(* CODESYS project EAS SCADA BATCH.library
   Company: ESCARRE AUTOMATIZACION Y SERVICIOS sl
   Description: Ajuste comunicacion ADS
      Ajuste tamaño constantes
   Version: 1.1.1
   Placeholder: EAS SCADA BATCH
   Author: EAS
   Title: EAS SCADA BATCH

Project tree, tasks and I/O mapping:
  libraries: Tc2_Standard, * (Beckhoff Automation GmbH); Tc2_System, * (Beckhoff Automation GmbH); Tc3_Module, * (Beckhoff Automation GmbH)
  DUTs/
    PE/
      data type E_Funcio
      data type PasCicle
      data type T_Compat
      data type T_funcio
      data type T_Sirena
  GVLs/
    global variables Batch
    global variables CONSTANTS
  POUs/
    BATCH/
      function block CarregarFuncionsActivesAlDB [ST]
      function block ComprobarFuncionsPas [ST]
      function block Inic_Func_Actv [ST]
      function block Parar_Func_FiFuncio [ST]
      function block Parar_Func_Incomp [ST]
      function block PararTotesLesFuncions [ST]
      function block Salt [ST]
      function block SaltDePasEnUnCicle [ST]
    GestioPE/
      function block FunBck_v01 [ST]
      function block Func_Activa_v01 [ST]
  VISUs/
*)

// DUTs/PE/E_Funcio
TYPE E_Funcio :
STRUCT

	Cd_Funcio:WORD;
	Actv_Funcio:BOOL;
	ParamFunc:ARRAY [1..Max_ParamFunc] OF WORD;

END_STRUCT
END_TYPE

// DUTs/PE/PasCicle
TYPE PasCicle :
STRUCT
	Pas:WORD;
	Funcio:E_Funcio;

END_STRUCT
END_TYPE

// DUTs/PE/T_Compat
TYPE T_Compat :
STRUCT

	Funcio1:WORD;  			(*Codi de la primera funcio*)
	Funcio2:WORD;  			(*Codi de la segona funcio*)

END_STRUCT
END_TYPE

// DUTs/PE/T_funcio
TYPE T_funcio :
STRUCT

	Cd_funcio:WORD;												(*Codi de la funció*)
	DesFuncio:STRING(16);										(*Descripció de la funció*)
	Background:BOOL;												(*Indicació per si la funció es en backgraund o no*)
	FinFunc:ARRAY [1..max_FinFunc] OF WORD;					(*Funcions que s'han d'acabar al començar aquesta*)

END_STRUCT
END_TYPE

// DUTs/PE/T_Sirena
TYPE T_Sirena :
STRUCT
	Actv:BOOL;
	Rearme:BOOL;
END_STRUCT
END_TYPE

// GVLs/Batch

VAR_GLOBAL RETAIN

(*=======================================	*)
(*					Estat del PE4							*)
(*=======================================	*)

(*Estat de PE4*)
	Func_Comp: ARRAY [1..Max_Compatibles] OF T_Compat;


(*=======================================	*)
(*			Variables de gestió de funcions				*)
(*=======================================	*)

(*Estat de lesFuncions *)
	Est_Func: ARRAY [1..Max_Funcions] OF E_Funcio;  		(*Estat actual de les funcions*)
	Est_F_PE4: ARRAY [1..Max_Funcions] OF E_Funcio;  		(*Estat de les funcions per les comunicacions del PE4*)
	Est_F_PE4_Ant: ARRAY [1..Max_Funcions] OF E_Funcio;  	(*Estat de les funcions per les comunicacions del PE4*)


(* *)
	Config_Func: ARRAY  [1..Max_Funcions] OF t_funcio;		(*Configuració de les funcios *)
	Func_Actives: ARRAY [1..Max_Func_Pas] OF WORD;		(* DB que indica en automaatic les funcions que estan en marcha en automatic*)


(*=======================================	*)
(*			Variables de gestió de cicle					*)
(*=======================================	*)

(*Cicles*)
	Cicle0: ARRAY [1..max_PasCicle] OF PasCicle;  			(*Cicle Actual de treball*)
	CicleRebut: ARRAY [1..max_PasCicle] OF PasCicle;  		(*Cicle Rebut*)


	

(*=======================================	*)
(*			Botons Auto/Man								*)
(*=======================================	*)

	PulsadorManual:BOOL;
	PulsadorAutomatic:BOOL;

(*=======================================	*)
(*			Marcas Internes								*)
(*=======================================	*)

	InicioCiclo:BOOL;


END_VAR


VAR_GLOBAL

(*=======================================	*)
(*			Maquina paralel 								*)
(*=======================================	*)

	TipoParalelo:WORD;
	MaquinaEnParalel:BOOL:=FALSE;
	Master:BOOL;
	Slave:BOOL;
	Pas_M:DWORD;
	Pas_S1:DWORD;
	Pas_S2:DWORD;
	Pas_S3:DWORD;
	Pas_S4:DWORD;
	Tipus_P:DWORD;
	Preparat_C_local:BOOL;
	He_C_local:BOOL;
	Ordre_C:BOOL;
	Ordre_C_Master:BOOL;
	Preparat_C_S1:BOOL;
	Preparat_C_S2:BOOL;
	Preparat_C_S3:BOOL;
	Preparat_C_S4:BOOL;
	He_C_S1:BOOL;
	He_C_S2:BOOL;
	He_C_S3:BOOL;
	He_C_S4:BOOL;
	Fi_C:BOOL;
	Fi_C_master:BOOL;



(*			CONSERVAR  COMPATIBILITAT				*)

	EsperaParalelPerSaltar:BOOL;
	SaltdePas:BOOL;


END_VAR

// GVLs/CONSTANTS

VAR_GLOBAL CONSTANT

(*=======================================	*)
(*			Carregar Constants						*)
(*=======================================	*)
	Max_Funcions:WORD:=128;
	Max_ParamFunc:WORD:=9;
	max_FinFunc:WORD:=5;
	max_PasCicle:WORD:=256;
	Max_Compatibles:WORD:=32;
	Max_Func_Pas:WORD:=12;

END_VAR


(*********************************************************************


	Max_ParamFixes:WORD:=150;
	Max_DBFiFuncio: WORD:=640 ;				(* Es calcula com    (Max_Funcions*Max_FinFunc)   *)
	Max_ElementsCicle: WORD:=2816 ;		(* Es calcula com    (Max_PasCicle*(Max_ParamFunc+2))  *)
	Max_DBIncompatibles: WORD:=128;			(* Es calcula com    (Max_Compatibles*2)  *)
	Max_Inputs: WORD:=128;
	Max_Outputs: WORD:=128;
	Max_Analog: WORD:=128;
	Num_Prod_Dos:WORD:=10;         					(* Numero maximo de productos en una dosificación*)
	Max_Prod_Dos:WORD:=128;							(* Productos en una dosificadora*)
	Max_Valv_Dos:WORD:=128;							(* Valvulas en una dosificadora*)
	Max_Alarmes:WORD:=128;



***************************************************************************)

// POUs/BATCH/CarregarFuncionsActivesAlDB
FUNCTION_BLOCK CarregarFuncionsActivesAlDB

(***********************************************************************
Aquest Bloc Carrega les Funcions actives al "DB d'estat de les funcions"
al "DB de funcions actives".   
************************************************************************)

VAR_INPUT
	EstatFuncions: ARRAY [1..max_funcions] OF E_Funcio;
END_VAR

VAR_OUTPUT
	FuncionsActives:ARRAY [1..Max_Func_Pas] OF WORD;
END_VAR

VAR
	Punter:WORD;
	PunterDB:WORD;
	inicialitzaDB: Inic_Func_Actv;
	DB_ple: BOOL;

END_VAR

inicialitzaDB(Func_Actv:= FuncionsActives);
DB_Ple:=FALSE;
punter:=1;
punterDB:=1;
WHILE (punter<=max_funcions)AND NOT(DB_Ple)
	DO
		IF EstatFuncions[punter].Actv_Funcio
			THEN
				FuncionsActives[PunterDB]:=EstatFuncions[punter].Cd_Funcio;
				PunterDB:=PunterDB+1;
				IF punterDB>Max_Func_Pas
					THEN
						DB_ple:=TRUE;
				END_IF
		END_IF
		punter:=punter+1;
END_WHILE

END_FUNCTION_BLOCK

// POUs/BATCH/Inic_Func_Actv
FUNCTION_BLOCK Inic_Func_Actv

(*********************************************************
Reinicia el DB de les funcions actives
***********************************************************)

VAR_IN_OUT
	Func_Actv: ARRAY [1..Max_Func_Pas] OF WORD;		(* DB que indica en automaatic les funcions que estan en marcha en automatic*)
END_VAR

VAR
	Punter: WORD;
END_VAR

Punter:=1;

REPEAT
	Func_Actv[punter]:=0;
	Punter:=Punter+1;
UNTIL
	Punter>Max_Func_Pas
END_REPEAT

END_FUNCTION_BLOCK

// POUs/BATCH/ComprobarFuncionsPas
FUNCTION_BLOCK ComprobarFuncionsPas

(************************************************************
Aquest Bloc Comproba les funcions actves que hi ha en aquest
pas i quan acaben dona l'ordr de canviar de pas.
**************************************************************)

VAR_INPUT
	Estat_F: ARRAY [1..Max_Funcions] OF E_Funcio;
	Tipus_F:ARRAY [1..Max_Funcions] OF T_Funcio;
	FuncionsActives:ARRAY [1..Max_Func_Pas] OF WORD;
END_VAR

VAR_OUTPUT
	AumentaPas:BOOL;
END_VAR

VAR
	Punter: WORD;
	Aumenta: BOOL;
	TempoPAS:TON;

END_VAR

(*Inicialitzar els punters*)
Punter:=1;
Aumenta:=TRUE;

REPEAT
	IF (FuncionsActives[Punter]<>0)AND((Estat_F[FuncionsActives[Punter]].Actv_Funcio=TRUE)AND(Tipus_F[FuncionsActives[Punter]].Background=FALSE))
		THEN
			Aumenta:=FALSE;
	END_IF
	Punter:=Punter+1;
UNTIL
	(Punter>Max_Func_Pas)OR(Aumenta=FALSE)
END_REPEAT

TempoPAS
	(IN:=Aumenta ,
	PT:=t#500ms ,
	Q=>AumentaPas ,
	ET=> );

END_FUNCTION_BLOCK

// POUs/BATCH/Parar_Func_FiFuncio
FUNCTION_BLOCK Parar_Func_FiFuncio

(**************************************************
Para les funcions del "DB de l'estat de funcions" 
depenen de la funcio de la entreda per "fifuncion"
***************************************************)

VAR_INPUT
	Tipus_Funcio:T_funcio;
END_VAR
VAR_OUTPUT
END_VAR
VAR_IN_OUT
	Estat_F: ARRAY [1..Max_Funcions] OF E_Funcio;
END_VAR
VAR
	PunterFiFunc:WORD;
	FuncioIncompat: WORD;
END_VAR

(*..................	Parar les funcions per fin función..................................	*)
PunterFiFunc:=1;
WHILE (PunterFiFunc <= max_FinFunc) DO
	FuncioIncompat :=Tipus_funcio.FinFunc[PunterFiFunc];
	IF FuncioIncompat <>0
		THEN
			Estat_F [FuncioIncompat].Actv_Funcio:=FALSE;
	END_IF
	PunterFiFunc:=PunterFiFunc+1;
END_WHILE

END_FUNCTION_BLOCK

// POUs/BATCH/Parar_Func_Incomp
FUNCTION_BLOCK Parar_Func_Incomp
(************************************************************
L'hi introduim una funció i el el bloc para les funcions del 
"DB estat de les funcions" depenen del 
"DB de compatibilitat"
**************************************************************)
VAR_INPUT
	Funcio:WORD;  (*Funcio que s'ha de parar*)
END_VAR

VAR_OUTPUT
END_VAR

VAR_IN_OUT
	DB_Comp:ARRAY [1..Max_Compatibles] OF T_Compat;
	Estat_F: ARRAY [1..Max_Funcions] OF E_Funcio;
END_VAR

VAR
	PunterEstat:WORD;
	PunterComp:WORD;
END_VAR

(*Mirar si hi ha alguna funció incompatible amb la nova funció*)
PunterEstat:=1;
PunterComp:=1;
REPEAT
	IF DB_Comp[PunterComp].Funcio1=Funcio
		THEN
			PunterEstat:=DB_Comp[PunterComp].Funcio2;
			Estat_F[PunterEstat].Actv_Funcio:=FALSE;
	END_IF
	PunterComp:=PunterComp+1;
UNTIL
	(PunterComp>Max_Compatibles)
END_REPEAT

END_FUNCTION_BLOCK

// POUs/BATCH/PararTotesLesFuncions
FUNCTION_BLOCK PararTotesLesFuncions
(********************************************************
Parar totes les funcions del "DB estat"
*********************************************************)
VAR_IN_OUT
	Estat_F: ARRAY [1..Max_Funcions] OF E_Funcio;
END_VAR

VAR
	Punter: WORD;
END_VAR

(*Inicialitzar els punters*)
Punter:=1;


WHILE (Punter <= Max_Funcions) DO
	IF Estat_F[Punter].Actv_Funcio=TRUE
		THEN
			Estat_F [Punter].Actv_Funcio:=FALSE;
	END_IF
	Punter:=Punter+1;
END_WHILE

END_FUNCTION_BLOCK

// POUs/BATCH/Salt
FUNCTION_BLOCK Salt
(************************************************************
Salta del "Pas inicial" al "Pas Final"  del  "BDCicle"
**************************************************************)
VAR_INPUT
	PasInicial:DWORD;
	PasFinal:DWORD;
END_VAR

VAR_IN_OUT


END_VAR

VAR

	FIFuncio:Parar_Func_FiFuncio;
	Incompatibles:Parar_Func_Incomp;
	PunterCicle:WORD;					(* Aquest valor marca la popsició del db de cicle on estem independent del pas de cicle *)
	T_Func_Act:T_Funcio;				(* Funcio que indica el punterCicle *)

	codi: WORD;

	Est_Func_0: ARRAY [1..Max_Funcions] OF E_Funcio;  		(*Estat de les funcions a cero per reiniciar l'estat*)
END_VAR

(*,,,,,,,,,,,,,,,,,,,,Carregar la posició inicial depenen si es salta desde:
				el pas cero: carerega d'un cicle nou
				un pas en concret: salt sobre el cicle que ja està carregat ,,,,,,,,,,,,,,,,,,,,,  *)

IF PasInicial=0
	THEN
		(*Posar Punter al primer pas*)
		PunterCicle:=1;
		(*Inicialitzar el estat de les funcions*)
		Est_Func:=Est_Func_0;
	ELSE
		(*Buscar Punter Cicle del pas inicial*)
		PunterCicle:=0;
		REPEAT
			PunterCicle := PunterCicle+1;
		UNTIL
			(((Cicle0[PunterCicle].Pas=PasInicial)AND(Cicle0[PunterCicle+1].Pas<>PasInicial)) OR (PunterCicle>=max_PasCicle))
		END_REPEAT
		PunterCicle := PunterCicle+1;      (*02/06/05*)
END_IF

(*,,,,,,,,,,,,,,,,,,,,Bucle de control,,,,,,,,,,,,,,,,,,,,,,,,,,,,,,,,,,,,,,,,,,,,,,,,,,,,,,,,,,,,,	*)

REPEAT
(*.................. Carregar la funció del pas............................................. *)
		codi:=Cicle0[PunterCicle].Funcio.Cd_Funcio;
		IF codi<>0 THEN
		T_Func_Act:=Config_Func[codi];
		END_IF
(*..................	Parar les funcions incompatibles..................................	*)
		Incompatibles(
			Funcio:=T_Func_Act.Cd_funcio ,
			DB_Comp:= Func_Comp ,
			Estat_F:= Est_Func );

(*..................	Activar si es en Background ........................................	*)
		IF T_Func_Act.Background=TRUE
			THEN
				Est_Func[T_Func_Act.Cd_Funcio] := Cicle0[PunterCicle].Funcio ; 	(*Carregar parametres*)
				Est_Func[T_Func_Act.Cd_Funcio].Actv_Funcio:=TRUE;			(*Posar la funció en actiu*)
		END_IF

(*..................	Parar les funcions per fin función..................................	*)
		FiFuncio(
			Tipus_Funcio:=  T_Func_Act ,
			 Estat_F:=Est_Func	 );

(*,,,,,,,,,,,,,,,,,,	Activar funció,,,,,,,,,,,,,,,,,,,,,,,,,,,,,,,,,,,,,,,,,,,,,,,,,,,,,,,,,,,,,,,,,,,	*)
		IF Cicle0[PunterCicle].Pas = PasFinal
			THEN
				Est_Func[T_Func_Act.Cd_Funcio] := Cicle0[PunterCicle].Funcio ;	(*Carregar parametres*)
				Est_Func[T_Func_Act.Cd_Funcio].Actv_Funcio := TRUE;			(*Posar la funció en actiu*)
		END_IF

(*,,,,,,,,,,,,,,,,,,Aumentar el Punter del cicle,,,,,,,,,,,,,,,,,,,,,,,,,,,,,,,,,,,,,,,,,,	*)
		PunterCicle := PunterCicle+1;

UNTIL
	(((Cicle0[PunterCicle].Pas <> PasFinal)AND(Cicle0[PunterCicle-1].Pas = PasFinal))
	OR(PunterCicle>max_PasCicle)
	OR(Cicle0[PunterCicle-1].Funcio.Cd_Funcio=0))
END_REPEAT

END_FUNCTION_BLOCK

// POUs/BATCH/SaltDePasEnUnCicle
FUNCTION_BLOCK SaltDePasEnUnCicle
(************************************************************
Salta del "Pas inicial" al "Pas Final"  del  "BDCicle"
**************************************************************)
VAR_INPUT
	PasInicial:DWORD;
	PasFinal:DWORD;
END_VAR

VAR_IN_OUT


END_VAR

VAR

	FIFuncio:Parar_Func_FiFuncio;
	Incompatibles:Parar_Func_Incomp;
	PunterCicle:WORD;					(* Aquest valor marca la popsició del db de cicle on estem independent del pas de cicle *)
	T_Func_Act:T_Funcio;				(* Funcio que indica el punterCicle *)

	codi: WORD;

	Est_Func_0: ARRAY [1..Max_Funcions] OF E_Funcio;  		(*Estat de les funcions a cero per reiniciar l'estat*)
END_VAR

(*,,,,,,,,,,,,,,,,,,,,Carregar la posició inicial depenen si es salta desde:
				el pas cero: carerega d'un cicle nou
				un pas en concret: salt sobre el cicle que ja està carregat ,,,,,,,,,,,,,,,,,,,,,  *)

IF PasInicial=0
	THEN
		(*Posar Punter al primer pas*)
		PunterCicle:=1;
		(*Inicialitzar el estat de les funcions*)
		Est_Func:=Est_Func_0;
	ELSE
		(*Buscar Punter Cicle del pas inicial*)
		PunterCicle:=0;
		REPEAT
			PunterCicle := PunterCicle+1;
		UNTIL
			(((Cicle0[PunterCicle].Pas=PasInicial)AND(Cicle0[PunterCicle+1].Pas<>PasInicial)) OR (PunterCicle>=max_PasCicle))
		END_REPEAT
		PunterCicle := PunterCicle+1;      (*02/06/05*)
END_IF

(*,,,,,,,,,,,,,,,,,,,,Bucle de control,,,,,,,,,,,,,,,,,,,,,,,,,,,,,,,,,,,,,,,,,,,,,,,,,,,,,,,,,,,,,	*)

REPEAT
(*.................. Carregar la funció del pas............................................. *)
		codi:=Cicle0[PunterCicle].Funcio.Cd_Funcio;
		IF codi<>0 THEN
		T_Func_Act:=Config_Func[codi];
		END_IF
(*..................	Parar les funcions incompatibles..................................	*)
		Incompatibles(
			Funcio:=T_Func_Act.Cd_funcio ,
			DB_Comp:= Func_Comp ,
			Estat_F:= Est_Func );

(*..................	Activar si es en Background ........................................	*)
		IF T_Func_Act.Background=TRUE
			THEN
				Est_Func[T_Func_Act.Cd_Funcio] := Cicle0[PunterCicle].Funcio ; 	(*Carregar parametres*)
				Est_Func[T_Func_Act.Cd_Funcio].Actv_Funcio:=TRUE;			(*Posar la funció en actiu*)
		END_IF

(*..................	Parar les funcions per fin función..................................
		FiFuncio(
			Tipus_Funcio:=  T_Func_Act ,
			 Estat_F:=Est_Func	 );										*)

(*,,,,,,,,,,,,,,,,,,	Activar funció,,,,,,,,,,,,,,,,,,,,,,,,,,,,,,,,,,,,,,,,,,,,,,,,,,,,,,,,,,,,,,,,,,,	*)
		IF Cicle0[PunterCicle].Pas = PasFinal
			THEN
				Est_Func[T_Func_Act.Cd_Funcio] := Cicle0[PunterCicle].Funcio ;	(*Carregar parametres*)
				Est_Func[T_Func_Act.Cd_Funcio].Actv_Funcio := TRUE;			(*Posar la funció en actiu*)
		END_IF

(*,,,,,,,,,,,,,,,,,,Aumentar el Punter del cicle,,,,,,,,,,,,,,,,,,,,,,,,,,,,,,,,,,,,,,,,,,	*)
		PunterCicle := PunterCicle+1;

UNTIL
	(((Cicle0[PunterCicle].Pas <> PasFinal)AND(Cicle0[PunterCicle-1].Pas = PasFinal))
	OR(PunterCicle>max_PasCicle)
	OR(Cicle0[PunterCicle-1].Funcio.Cd_Funcio=0))
END_REPEAT

END_FUNCTION_BLOCK

// POUs/GestioPE/FunBck_v01
FUNCTION_BLOCK FunBck_v01
VAR_INPUT
END_VAR

VAR_OUTPUT
	funcioBck: BOOL;
END_VAR


VAR
	punter: WORD;
END_VAR

punter:=1;
funcioBck:=FALSE;

WHILE ((punter<= Max_Funcions)AND NOT(FuncioBck)) DO
	IF ((Est_func[punter].Actv_funcio)AND NOT(Config_Func[punter].Background))
		THEN
			FuncioBck:=TRUE;
	END_IF
	punter:=punter+1;
END_WHILE

END_FUNCTION_BLOCK

// POUs/GestioPE/Func_Activa_v01
FUNCTION_BLOCK Func_Activa_v01
VAR_INPUT
	EstatFunc:ARRAY [1..Max_Funcions] OF E_Funcio;
END_VAR
VAR_OUTPUT
	FuncionsActives:BOOL;
END_VAR
VAR
	a: WORD;
END_VAR

(*Inicialitza el punter*)
a:=1;
FuncionsActives:=FALSE;
REPEAT
	IF EstatFunc[a].Actv_Funcio=TRUE
		THEN
			FuncionsActives:=TRUE;
	END_IF
	a:=a+1;
UNTIL
(a>Max_Funcions)OR(FuncionsActives=TRUE)
END_REPEAT

END_FUNCTION_BLOCK
